{attribute 'call_after_init'}
FUNCTION_BLOCK FB_BaseplateChiller_Test EXTENDS FB_TestSuite
VAR_INPUT
END_VAR
VAR_OUTPUT
END_VAR
VAR
END_VAR

ErrorTriggers();
ErrorResets();
ErrorLatches();
NoError();

METHOD ErrorLatches
VAR
	fbBaseplateChiller : FB_BaseplateChiller := F_BaseplateChiller_Error();
END_VAR
TEST('ErrorLatches');

fbBaseplateChiller(bBaseplateChillerFlow := TRUE);
AssertTrue(fbBaseplateChiller.bError, 'Error did not latch');

TEST_FINISHED();
END_METHOD

METHOD ErrorResets
VAR
	fbBaseplateChiller : FB_BaseplateChiller := F_BaseplateChiller_Error();
END_VAR
TEST('ErrorResets');

fbBaseplateChiller.Reset();
fbBaseplateChiller(bBaseplateChillerFlow := TRUE);
AssertFalse(fbBaseplateChiller.bError, 'Error did not reset');

TEST_FINISHED();
END_METHOD

METHOD ErrorTriggers
VAR
	fbBaseplateChiller : FB_BaseplateChiller := F_BaseplateChiller_Error();
END_VAR
TEST('ErrorTriggers');

AssertTrue(fbBaseplateChiller.bError, 'Error did not trigger');

TEST_FINISHED();
END_METHOD

METHOD NoError
VAR
	fbBaseplateChiller : FB_BaseplateChiller;
END_VAR
TEST('NoError');

fbBaseplateChiller(bBaseplateChillerFlow := TRUE);
AssertFalse(fbBaseplateChiller.bError, 'Error falsely triggered');

TEST_FINISHED();
END_METHOD

END_FUNCTION_BLOCK

(* stored: Version 1.1.0.1, ProductVersion 3.1.4020.14
   POU FB_BaseplateChiller_Test: Id {572d3bba-8454-4f82-8787-2e97fb394969}, SpecialFunc None
   Method ErrorLatches: Id {58214f70-e372-4736-8bfc-f1749ed7fbb3}
   Method ErrorResets: Id {32fb2b02-0dbd-48f4-ac77-6d502573fb17}
   Method ErrorTriggers: Id {e75ff8cd-5e84-4dec-b552-f9030ddf8e8a}
   Method NoError: Id {6c8e266e-98ed-4819-a029-9292e0cd29ec} *)
